(* IEC 61131-3 sources: ST2CPP/examples/projects/smart_factory, 7 files *)

(* ---- types.st ---- *)
(* smart_factory/types.st — 类型定义 *)

(* 传感器数据包 *)
TYPE SENSOR_DATA :
STRUCT
    TEMPERATURE : REAL;
    HUMIDITY    : REAL;
    PRESSURE    : REAL;
    LIGHT       : INT;
END_STRUCT;
END_TYPE

(* 电机状态 *)
TYPE MOTOR_STATUS :
STRUCT
    SPEED       : INT;
    TORQUE      : REAL;
    DIRECTION   : INT;       (* 0=停止, 1=正转, 2=反转 *)
    ERROR_CODE  : INT;
END_STRUCT;
END_TYPE

(* 报警级别 *)
TYPE ALARM_LEVEL : (NONE, LOW, MEDIUM, HIGH, CRITICAL);
END_TYPE

(* 配方参数 *)
TYPE RECIPE :
STRUCT
    TEMP_TARGET   : REAL;
    TIME_SECONDS  : INT;
    SPEED_SET     : INT;
    TOLERANCE     : REAL;
END_STRUCT;
END_TYPE

(* ---- utils.st ---- *)
(* smart_factory/utils.st — 工具函数 *)

FUNCTION CLAMP_INT : DINT
    VAR_INPUT
        VAL  : DINT;
        MINV : DINT;
        MAXV : DINT;
    END_VAR
    IF VAL < MINV THEN
        CLAMP_INT := MINV;
    ELSIF VAL > MAXV THEN
        CLAMP_INT := MAXV;
    ELSE
        CLAMP_INT := VAL;
    END_IF
END_FUNCTION

FUNCTION SCALE_REAL : REAL
    VAR_INPUT
        INPUT_VAL : REAL;
        IN_MIN    : REAL;
        IN_MAX    : REAL;
        OUT_MIN   : REAL;
        OUT_MAX   : REAL;
    END_VAR
    VAR
        RATIO : REAL;
    END_VAR
    IF IN_MAX = IN_MIN THEN
        SCALE_REAL := OUT_MIN;
    ELSE
        RATIO := (INPUT_VAL - IN_MIN) / (IN_MAX - IN_MIN);
        SCALE_REAL := OUT_MIN + RATIO * (OUT_MAX - OUT_MIN);
    END_IF
END_FUNCTION

FUNCTION BIT_CHECK : BOOL
    VAR_INPUT
        VALUE : INT;
        BIT_POS : INT;
    END_VAR
    VAR
        MASK : INT;
    END_VAR
    MASK := 1;
    IF BIT_POS > 0 THEN
        MASK := SHL(MASK, BIT_POS);
    END_IF
    IF (VALUE AND MASK) <> 0 THEN
        BIT_CHECK := TRUE;
    ELSE
        BIT_CHECK := FALSE;
    END_IF
END_FUNCTION

FUNCTION WRAP_ANGLE : INT
    VAR_INPUT
        ANGLE : INT;
    END_VAR
    WHILE ANGLE < 0 DO
        ANGLE := ANGLE + 360;
    END_WHILE
    WHILE ANGLE >= 360 DO
        ANGLE := ANGLE - 360;
    END_WHILE
    WRAP_ANGLE := ANGLE;
END_FUNCTION

(* ---- base_controller.st ---- *)
(* smart_factory/base_controller.st — 基础控制器 CLASS *)

CLASS BASE_CONTROLLER
    VAR
        SYSTEM_STATE  : INT := 0;
        CYCLE_COUNT   : DINT := 0;
        RUN_ENABLE    : BOOL := FALSE;
    END_VAR

    METHOD STARTUP : BOOL
        RUN_ENABLE := TRUE;
        SYSTEM_STATE := 1;
        STARTUP := TRUE;
    END_METHOD

    METHOD SHUTDOWN : BOOL
        RUN_ENABLE := FALSE;
        SYSTEM_STATE := 0;
        SHUTDOWN := TRUE;
    END_METHOD

    METHOD GET_STATE : INT
        GET_STATE := SYSTEM_STATE;
    END_METHOD

    METHOD TICK
        IF RUN_ENABLE THEN
            CYCLE_COUNT := CYCLE_COUNT + 1;
        END_IF
    END_METHOD
END_CLASS

(* ---- line_controller.st ---- *)
(* smart_factory/line_controller.st — 产线控制器 CLASS *)

CLASS LINE_CONTROLLER
    VAR
        LINE_ID       : INT := 0;
        PROD_COUNT    : DINT := 0;
        RUN_ENABLE    : BOOL := FALSE;
    END_VAR

    METHOD INIT_LINE : BOOL
        RUN_ENABLE := TRUE;
        LINE_ID := 1;
        PROD_COUNT := 0;
        INIT_LINE := TRUE;
    END_METHOD

    METHOD PROD_CYCLE : DINT
        IF RUN_ENABLE THEN
            PROD_COUNT := PROD_COUNT + 1;
        END_IF
        PROD_CYCLE := PROD_COUNT;
    END_METHOD
END_CLASS

(* ---- motor_ctrl.st ---- *)
(* smart_factory/motor_ctrl.st — 电机控制 FB *)

FUNCTION_BLOCK MOTOR_CTRL
    VAR_INPUT
        ENABLE      : BOOL;
        TARGET_SPEED : INT;
        CMD_DIR     : INT;       (* 0=停止, 1=正转, 2=反转 *)
    END_VAR
    VAR_OUTPUT
        STATUS      : MOTOR_STATUS;
        ACTUAL_SPEED : INT;
        IS_RUNNING  : BOOL;
    END_VAR
    VAR
        RAMP_STEP   : INT := 10;
        CURRENT_SPD : INT := 0;
        ERROR       : INT := 0;
    END_VAR

    IS_RUNNING := ENABLE AND (CMD_DIR <> 0);

    IF NOT ENABLE OR CMD_DIR = 0 THEN
        (* 停车：减速 *)
        IF CURRENT_SPD > 0 THEN
            CURRENT_SPD := CURRENT_SPD - RAMP_STEP;
            IF CURRENT_SPD < 0 THEN
                CURRENT_SPD := 0;
            END_IF
        ELSIF CURRENT_SPD < 0 THEN
            CURRENT_SPD := CURRENT_SPD + RAMP_STEP;
            IF CURRENT_SPD > 0 THEN
                CURRENT_SPD := 0;
            END_IF
        END_IF
    ELSE
        (* 加速到目标 *)
        IF CURRENT_SPD < TARGET_SPEED THEN
            CURRENT_SPD := CURRENT_SPD + RAMP_STEP;
            IF CURRENT_SPD > TARGET_SPEED THEN
                CURRENT_SPD := TARGET_SPEED;
            END_IF
        ELSIF CURRENT_SPD > TARGET_SPEED THEN
            CURRENT_SPD := CURRENT_SPD - RAMP_STEP;
            IF CURRENT_SPD < TARGET_SPEED THEN
                CURRENT_SPD := TARGET_SPEED;
            END_IF
        END_IF
    END_IF
    ACTUAL_SPEED := CURRENT_SPD;

    (* 填充状态 *)
    STATUS.SPEED := CURRENT_SPD;
    STATUS.TORQUE := REAL#0.0;
    STATUS.DIRECTION := CMD_DIR;
    STATUS.ERROR_CODE := ERROR;
END_FUNCTION_BLOCK

(* ---- sensor_ctrl.st ---- *)
(* smart_factory/sensor_ctrl.st — 传感器控制 FB *)

FUNCTION_BLOCK SENSOR_CTRL
    VAR_INPUT
        ENABLE      : BOOL;
        RAW_TEMP    : REAL;
        RAW_HUMID   : REAL;
        RAW_PRESS   : REAL;
        RAW_LIGHT   : INT;
    END_VAR
    VAR_OUTPUT
        DATA        : SENSOR_DATA;
        ALARM       : ALARM_LEVEL;
        FILTERED_OK : BOOL;
    END_VAR
    VAR
        SAMPLE_COUNT : DINT := 0;
        SUM_TEMP     : REAL := 0.0;
        SUM_HUMID    : REAL := 0.0;
        BASE_TEMP    : REAL := 25.0;
    END_VAR

    IF NOT ENABLE THEN
        FILTERED_OK := FALSE;
        ALARM := ALARM_LEVEL#NONE;
        RETURN;
    END_IF

    (* 累加采样 *)
    SAMPLE_COUNT := SAMPLE_COUNT + 1;
    SUM_TEMP := SUM_TEMP + RAW_TEMP;
    SUM_HUMID := SUM_HUMID + RAW_HUMID;

    (* 输出原始数据 *)
    DATA.TEMPERATURE := RAW_TEMP;
    DATA.HUMIDITY := RAW_HUMID;
    DATA.PRESSURE := RAW_PRESS;
    DATA.LIGHT := RAW_LIGHT;

    (* 简单滤波判断 *)
    FILTERED_OK := TRUE;

    (* 温度报警 *)
    IF RAW_TEMP > 80.0 THEN
        ALARM := ALARM_LEVEL#HIGH;
        FILTERED_OK := FALSE;
    ELSIF RAW_TEMP > 60.0 THEN
        ALARM := ALARM_LEVEL#MEDIUM;
    ELSIF RAW_TEMP < 0.0 THEN
        ALARM := ALARM_LEVEL#LOW;
    ELSE
        ALARM := ALARM_LEVEL#NONE;
    END_IF
END_FUNCTION_BLOCK

(* ---- main.st ---- *)
(* smart_factory/main.st — 主程序 *)

PROGRAM SMART_FACTORY_MAIN
    VAR
        Sensor      : SENSOR_CTRL;
        SensorData  : SENSOR_DATA;
        SensorAlarm : ALARM_LEVEL;
        SensorOK    : BOOL := FALSE;

        Motor       : MOTOR_CTRL;
        MotorStatus : MOTOR_STATUS;
        MotorSpeed  : INT := 0;
        MotorRunning : BOOL := FALSE;

        LineCtrl    : LINE_CONTROLLER;
        LineProd    : DINT := 0;

        CurrentRecipe : RECIPE;

        CYCLE       : DINT := 0;
        STOP_CMD    : BOOL := FALSE;

        RAW_T   : REAL := 25.0;
        RAW_H   : REAL := 50.0;
        RAW_P   : REAL := 1013.0;
        RAW_L   : INT := 500;

        SPD_CMD : INT := 1000;
        DIR_CMD : INT := 1;

        WRAPPED : INT := 0;
        SCALED  : REAL := 0.0;
        BIT_VAL : INT := 16#00FF;
        BIT_OK  : BOOL := FALSE;

        INIT_DONE : BOOL := FALSE;
    END_VAR

    IF NOT INIT_DONE THEN
        LineCtrl.INIT_LINE();
        INIT_DONE := TRUE;
        CurrentRecipe.TEMP_TARGET := 85.0;
        CurrentRecipe.TIME_SECONDS := 300;
        CurrentRecipe.SPEED_SET := 1500;
        CurrentRecipe.TOLERANCE := 0.5;
        PRINT("=== SMART FACTORY START ===");
    END_IF

    LineProd := LineCtrl.PROD_CYCLE();

    WRAPPED := WRAP_ANGLE(ANGLE := 450);
    ASSERT(WRAPPED = 90);

    SCALED := SCALE_REAL(INPUT_VAL := 50.0, IN_MIN := 0.0, IN_MAX := 100.0, OUT_MIN := 0.0, OUT_MAX := 270.0);

    BIT_OK := BIT_CHECK(VALUE := BIT_VAL, BIT_POS := 3);
    ASSERT(BIT_OK = TRUE);

    Sensor(
        ENABLE := TRUE,
        RAW_TEMP := RAW_T,
        RAW_HUMID := RAW_H,
        RAW_PRESS := RAW_P,
        RAW_LIGHT := RAW_L,
        DATA => SensorData,
        ALARM => SensorAlarm,
        FILTERED_OK => SensorOK
    );

    Motor(
        ENABLE := TRUE,
        TARGET_SPEED := SPD_CMD,
        CMD_DIR := DIR_CMD,
        STATUS => MotorStatus,
        ACTUAL_SPEED => MotorSpeed,
        IS_RUNNING => MotorRunning
    );

    IF (BIT_VAL AND 16#0010) <> 0 THEN
        PRINT("BIT 4 is set");
    END_IF

    IF (BIT_VAL OR 16#FF00) = 16#FFFF THEN
        PRINT("OR mask OK");
    END_IF

    ASSERT(LineProd >= 0);
    ASSERT(SensorOK = TRUE);
    ASSERT(MotorSpeed > 0);
    ASSERT(MotorRunning = TRUE);
    ASSERT(SensorData.TEMPERATURE = 25.0);
    ASSERT(CurrentRecipe.TEMP_TARGET = 85.0);

    CYCLE := CYCLE + 1;
    PRINT("CYCLE=" + CYCLE + " PROD=" + LineProd + " SPD=" + MotorSpeed);
END_PROGRAM
